{attribute 'GeneratedUsingTerminal: IODEVICETYPE_ETHERCATPROT'}
{attribute addProperty BoxType "IODEVICETYPE_ETHERCATPROT"}
{attribute addProperty Id "EK1100_Beckhoff_AMI8xxxEK1100_Beckhoff_AMI8xxx_7CB3D10B80SyncUnitsSyncUnits_3DFA47ED27InputsInputs_25A0042B160OutputsOutputs_2397A10E106InfoDataInfoData_E68C61CD28"}
{attribute addProperty CRC "3472833195"}
{attribute addProperty Size "401"}
TYPE EtherCAT_Master_AMIxxxx_CEFF3AAB :
STRUCT
	{attribute addProperty Name "EK1100_Beckhoff_AMI8xxx"}
	{attribute addProperty PreviousPort "EtherCAT_Master_AMIxxxx : Master"}
	EK1100_Beckhoff_AMI8xxx : EK1100_Beckhoff_AMI8xxx_7CB3D10B;
	{attribute addProperty Name "SyncUnits"}
	SyncUnits : SyncUnits_3DFA47ED;
	{attribute addProperty Name "Inputs"}
	Inputs : Inputs_25A0042B;
	{attribute addProperty Name "Outputs"}
	Outputs : Outputs_2397A10E;
	{attribute addProperty Name "InfoData"}
	InfoData : InfoData_E68C61CD;
END_STRUCT
END_TYPE

(* stored: Version 1.2.0.0, ProductVersion 3.1.4024.9
   DUT EtherCAT_Master_AMIxxxx_CEFF3AAB: Id {1ee902ed-f75d-411a-bcb5-51a66bc24699} *)
